FUNCTION_BLOCK FB_SimCheckWeigher EXTENDS FB_SimStation
VAR_INPUT
END_VAR
VAR_OUTPUT
END_VAR
VAR	
	tmrWork						: TON;
END_VAR

METHOD PROTECTED  DoWork : BOOL
VAR_INPUT
END_VAR
tmrWork(IN:=TRUE, PT:=T#2S);
IF tmrWork.Q THEN
	tmrWork(IN:=FALSE);
	DoWork := TRUE;
END_IF
END_METHOD

METHOD PROTECTED  UpdatePartStatus : PVOID
VAR_INPUT
END_VAR
IF pPartStatus <> 0 THEN
	pPartStatus^.bWeightStatus := TRUE;
	pPartStatus^.fActualWeightMg := 100;
END_IF
END_METHOD

END_FUNCTION_BLOCK

(* stored: Version 1.1.0.1, ProductVersion 3.1.4024.12
   POU FB_SimCheckWeigher: Id {6e33866b-3474-4e96-8cf0-c26d69bfb058}, SpecialFunc None
   Method DoWork: Id {71bfd5a5-86f3-4639-9c36-fd5ab9d1fe15}
   Method UpdatePartStatus: Id {0a54fb0a-f4e0-450f-814a-141a3dd7ad3e} *)
